(* Logix 5000 project; controller GEA_Test_Chamber vendor 1 type 14 code 196 rev 32.14; software revision 32.04; part 8 of 11 *)
(* tags used below, declared in another part *)
   Act_Time : DINT[7];
   Actuators_OnOff_Heater : BOOL;
   bPulse10Hz : BOOL;
   bPulse1Hz : BOOL;
   Counter : COUNTER[20];
   DRK375_Flow_Change : BOOL;
   DRK375_Flow_InRange : BOOL;
   DRK375_Temp_Change : BOOL;
   DRK375_Temp_InRange : BOOL;
   Flow_Change_Step : INT;
   FVIR_Water_DRK375_Error : REAL;
   Heater_OnOff : BOOL;
   LDO_DRK375_Start : BOOL;
   LDO_LabView_Comm_OK : BOOL;
   LDO_Step : INT;
   LDO_TestFlow : BOOL;
   LDO_Timer_Delay : TIMER[30];
   LDO_Water_float : REAL;
   LDO_Water_Flow_DRK375_REG : REAL;
   LDO_Water_Flow_DRK375_SP : INT;
   LDO_Water_SP_float : REAL;
   LDO_Water_Temp_DRK375_SP : INT;
   LDO_Water_Temp_float : REAL;
   LDO_Water_Temp_SP_float : REAL;
   LDO_WaterHeater_Step : INT;
   New_Time : BOOL;
   ONS : BOOL[32];
   puls_start : BOOL;
   puls_stop : BOOL;
   Pulse : BOOL[32];
   T_Diff_WaterStep10 : T_DIFF;
   T_Diff_WaterStep20 : T_DIFF;
   T_Diff_WaterStep40 : T_DIFF;
   T_Diff_WaterStep50 : T_DIFF;
   T_Diff_WaterStep70 : T_DIFF;
   T_Diff_WaterStep80 : T_DIFF;
   Temp_Change_Step : INT;
   Timer_Delay : TIMER[30];
   Water_Flow_Calc_float : REAL;
   Water_Flow_DRK375 : INT;
   Water_Outlet_InRange_LDO : BOOL;
   Water_Step_10 : DINT[7];
   Water_Step_10_Done : BOOL;
   Water_Step_20 : DINT[7];
   Water_Step_20_Done : BOOL;
   Water_Step_401 : DINT[7];
   Water_Step_40_Done : BOOL;
   Water_Step_50 : DINT[7];
   Water_Step_50_Done : BOOL;
   Water_Step_70 : DINT[7];
   Water_Step_70_Done : BOOL;
   Water_Step_80 : DINT[7];
   Water_Step_80_Done : BOOL;
   Water_T_Diff_10 : DINT;
   Water_T_Diff_20 : DINT;
   Water_T_Diff_40 : DINT;
   Water_T_Diff_50 : DINT;
   Water_T_Diff_70 : DINT;
   Water_T_Diff_80 : DINT;
   Water_Temp_Calc_float : REAL;
   Water_Temp_DRK375 : INT;
   Water_Temp_DRK375_Last : REAL;
   Heater_Cnt : COUNTER;
   LDO_Error_MSG : INT;
   LDO_LabView_Control : INT;
   LDO_Water_Flow_DRK375_Float : REAL;
   LDO_Water_Temp_DRK375_Float : REAL;
   Output_LDO : Output_LDO;
   Water_Flow_DRK375_Last_Float : REAL;
(* LDO_Chamber, continued *)

ROUTINE LDO_Error_MSG   (* ladder *)
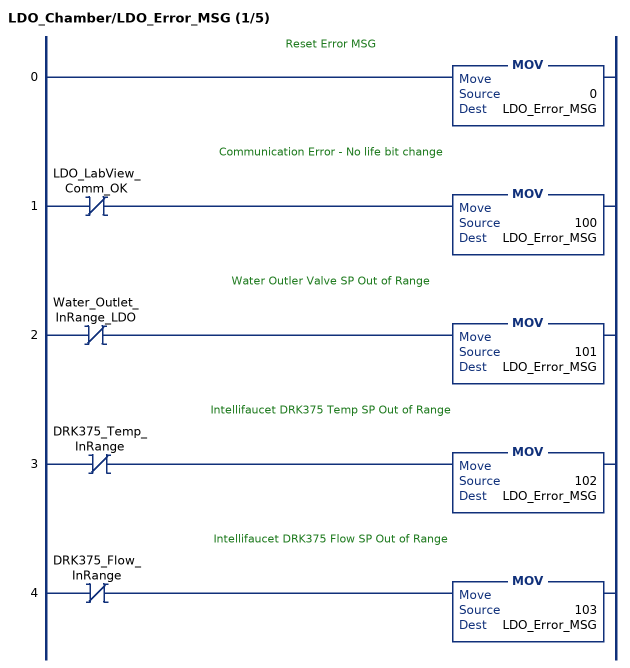
   // Reset Error MSG
   0: MOV(0,LDO_Error_MSG);
   // Communication Error - No life bit change
   1: XIO(LDO_LabView_Comm_OK)MOV(100,LDO_Error_MSG);
   // Water Outler Valve SP Out of Range
   2: XIO(Water_Outlet_InRange_LDO)MOV(101,LDO_Error_MSG);
   // Intellifaucet DRK375 Temp SP Out of Range
   3: XIO(DRK375_Temp_InRange)MOV(102,LDO_Error_MSG);
   // Intellifaucet DRK375 Flow SP Out of Range
   4: XIO(DRK375_Flow_InRange)MOV(103,LDO_Error_MSG);
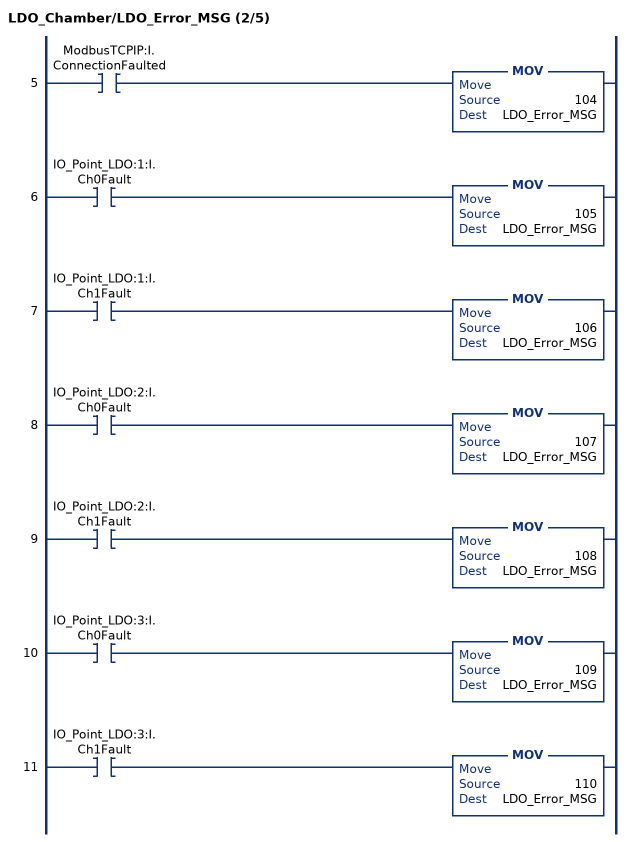
   5: XIC(ModbusTCPIP:I.ConnectionFaulted)MOV(104,LDO_Error_MSG);
   6: XIC(IO_Point_LDO:1:I.Ch0Fault)MOV(105,LDO_Error_MSG);
   7: XIC(IO_Point_LDO:1:I.Ch1Fault)MOV(106,LDO_Error_MSG);
   8: XIC(IO_Point_LDO:2:I.Ch0Fault)MOV(107,LDO_Error_MSG);
   9: XIC(IO_Point_LDO:2:I.Ch1Fault)MOV(108,LDO_Error_MSG);
   10: XIC(IO_Point_LDO:3:I.Ch0Fault)MOV(109,LDO_Error_MSG);
   11: XIC(IO_Point_LDO:3:I.Ch1Fault)MOV(110,LDO_Error_MSG);
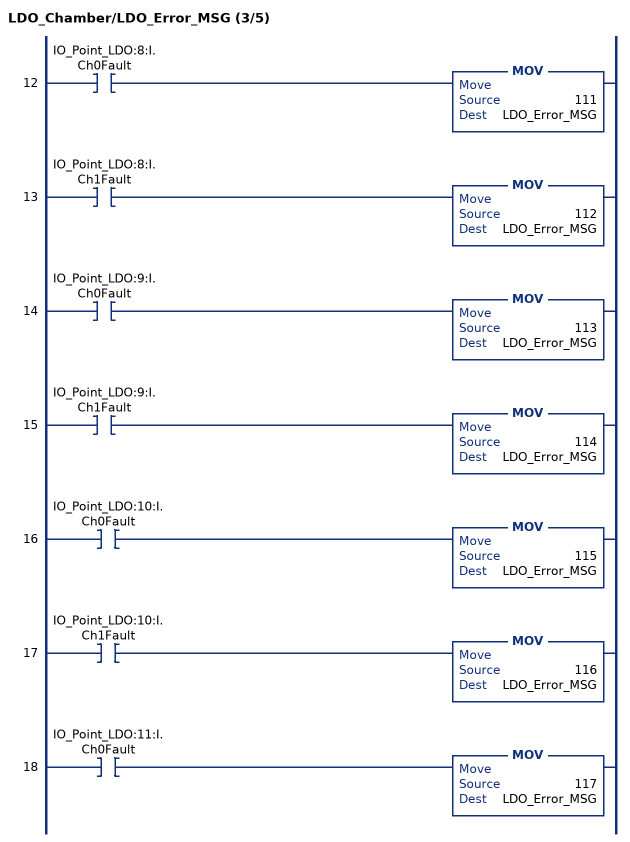
   12: XIC(IO_Point_LDO:8:I.Ch0Fault)MOV(111,LDO_Error_MSG);
   13: XIC(IO_Point_LDO:8:I.Ch1Fault)MOV(112,LDO_Error_MSG);
   14: XIC(IO_Point_LDO:9:I.Ch0Fault)MOV(113,LDO_Error_MSG);
   15: XIC(IO_Point_LDO:9:I.Ch1Fault)MOV(114,LDO_Error_MSG);
   16: XIC(IO_Point_LDO:10:I.Ch0Fault)MOV(115,LDO_Error_MSG);
   17: XIC(IO_Point_LDO:10:I.Ch1Fault)MOV(116,LDO_Error_MSG);
   18: XIC(IO_Point_LDO:11:I.Ch0Fault)MOV(117,LDO_Error_MSG);
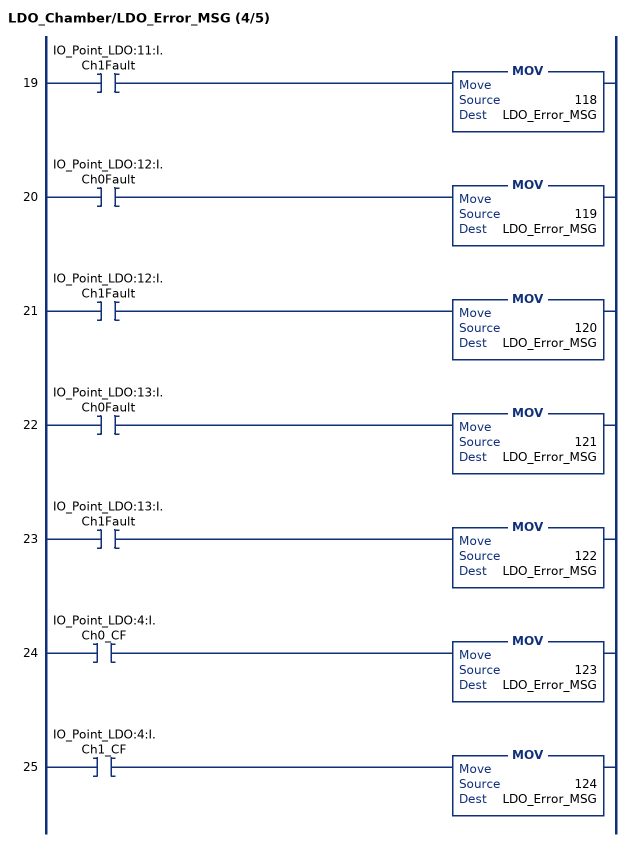
   19: XIC(IO_Point_LDO:11:I.Ch1Fault)MOV(118,LDO_Error_MSG);
   20: XIC(IO_Point_LDO:12:I.Ch0Fault)MOV(119,LDO_Error_MSG);
   21: XIC(IO_Point_LDO:12:I.Ch1Fault)MOV(120,LDO_Error_MSG);
   22: XIC(IO_Point_LDO:13:I.Ch0Fault)MOV(121,LDO_Error_MSG);
   23: XIC(IO_Point_LDO:13:I.Ch1Fault)MOV(122,LDO_Error_MSG);
   24: XIC(IO_Point_LDO:4:I.Ch0_CF)MOV(123,LDO_Error_MSG);
   25: XIC(IO_Point_LDO:4:I.Ch1_CF)MOV(124,LDO_Error_MSG);
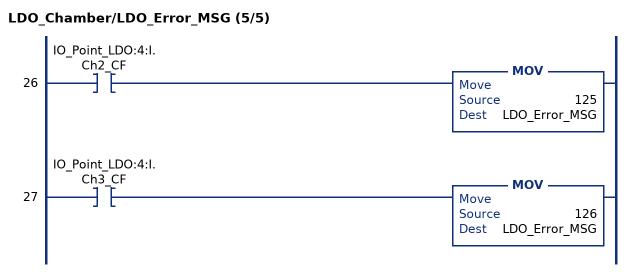
   26: XIC(IO_Point_LDO:4:I.Ch2_CF)MOV(125,LDO_Error_MSG);
   27: XIC(IO_Point_LDO:4:I.Ch3_CF)MOV(126,LDO_Error_MSG);
END_ROUTINE

ROUTINE LDO_Heater_OnOff   (* ladder *)
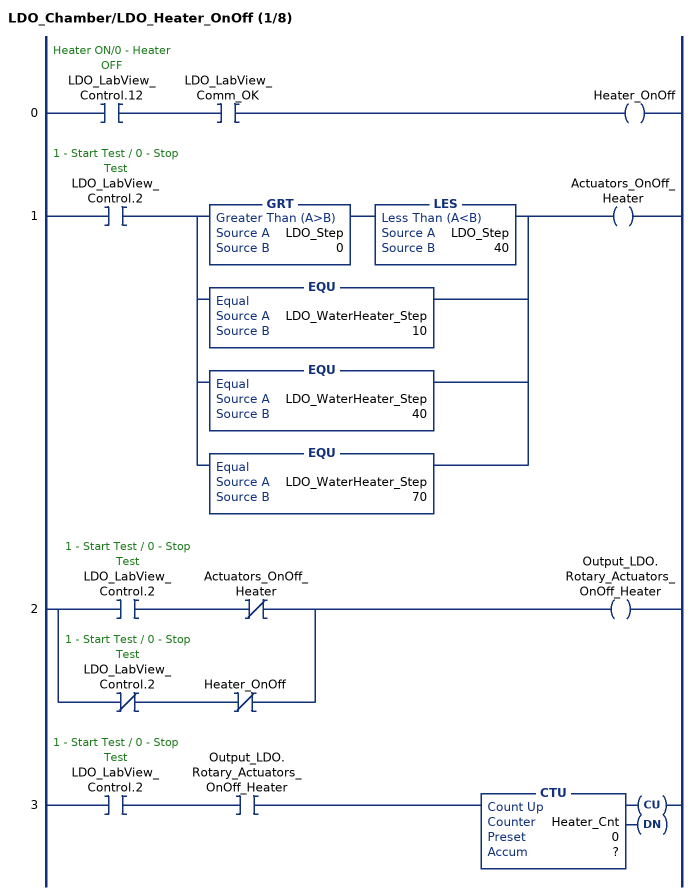
   0: XIC(LDO_LabView_Control.12)XIC(LDO_LabView_Comm_OK)OTE(Heater_OnOff);
   1: XIC(LDO_LabView_Control.2)[GRT(LDO_Step,0) LES(LDO_Step,40) ,EQU(LDO_WaterHeater_Step,10) ,EQU(LDO_WaterHeater_Step,40) ,EQU(LDO_WaterHeater_Step,70) ]OTE(Actuators_OnOff_Heater);
   2: [XIC(LDO_LabView_Control.2) XIO(Actuators_OnOff_Heater) ,XIO(LDO_LabView_Control.2) XIO(Heater_OnOff) ]OTE(Output_LDO.Rotary_Actuators_OnOff_Heater);
   3: XIC(LDO_LabView_Control.2)XIC(Output_LDO.Rotary_Actuators_OnOff_Heater)CTU(Heater_Cnt,?,?);
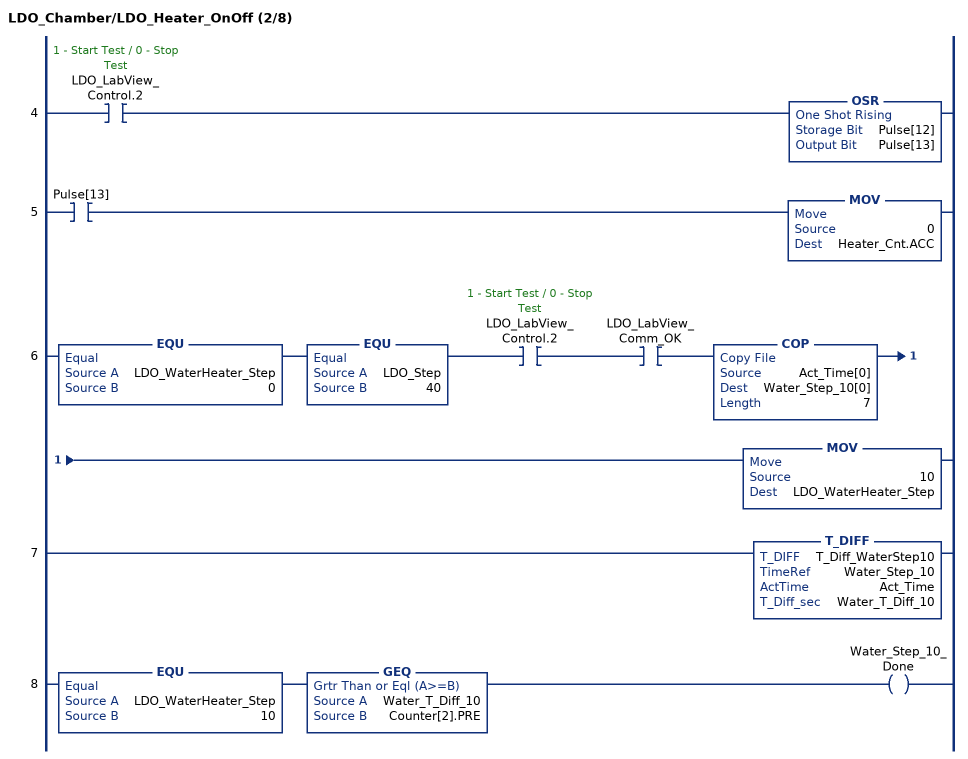
   4: XIC(LDO_LabView_Control.2)OSR(Pulse[12],Pulse[13]);
   5: XIC(Pulse[13])MOV(0,Heater_Cnt.ACC);
   6: EQU(LDO_WaterHeater_Step,0)EQU(LDO_Step,40)XIC(LDO_LabView_Control.2)XIC(LDO_LabView_Comm_OK)COP(Act_Time[0],Water_Step_10[0],7)MOV(10,LDO_WaterHeater_Step);
   7: T_DIFF(T_Diff_WaterStep10,Water_Step_10,Act_Time,Water_T_Diff_10);
   8: EQU(LDO_WaterHeater_Step,10)GEQ(Water_T_Diff_10,Counter[2].PRE)OTE(Water_Step_10_Done);
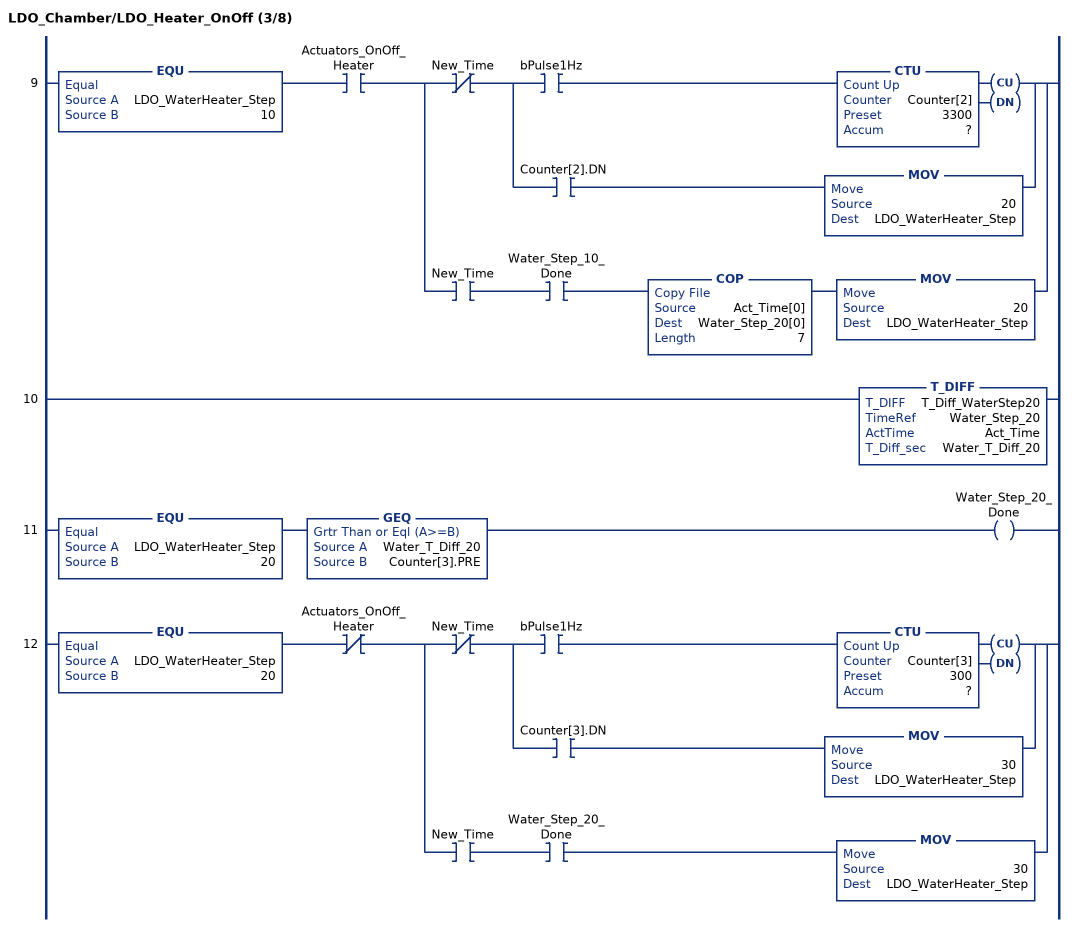
   9: EQU(LDO_WaterHeater_Step,10)XIC(Actuators_OnOff_Heater)[XIO(New_Time) [XIC(bPulse1Hz) CTU(Counter[2],?,?) ,XIC(Counter[2].DN) MOV(20,LDO_WaterHeater_Step) ] ,XIC(New_Time) XIC(Water_Step_10_Done) COP(Act_Time[0],Water_Step_20[0],7) MOV(20,LDO_WaterHeater_Step) ];
   10: T_DIFF(T_Diff_WaterStep20,Water_Step_20,Act_Time,Water_T_Diff_20);
   11: EQU(LDO_WaterHeater_Step,20)GEQ(Water_T_Diff_20,Counter[3].PRE)OTE(Water_Step_20_Done);
   12: EQU(LDO_WaterHeater_Step,20)XIO(Actuators_OnOff_Heater)[XIO(New_Time) [XIC(bPulse1Hz) CTU(Counter[3],?,?) ,XIC(Counter[3].DN) MOV(30,LDO_WaterHeater_Step) ] ,XIC(New_Time) XIC(Water_Step_20_Done) MOV(30,LDO_WaterHeater_Step) ];
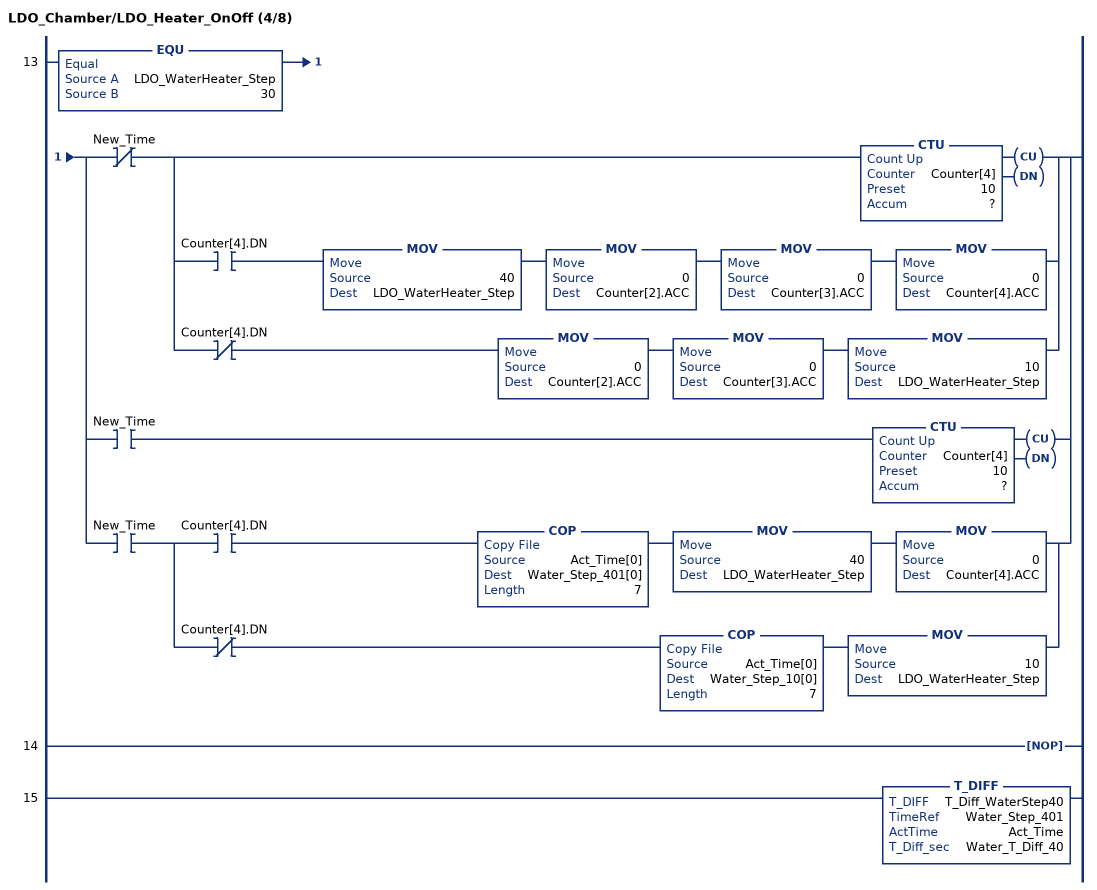
   13: EQU(LDO_WaterHeater_Step,30)[XIO(New_Time) [CTU(Counter[4],?,?) ,XIC(Counter[4].DN) MOV(40,LDO_WaterHeater_Step) MOV(0,Counter[2].ACC) MOV(0,Counter[3].ACC) MOV(0,Counter[4].ACC) ,XIO(Counter[4].DN) MOV(0,Counter[2].ACC) MOV(0,Counter[3].ACC) MOV(10,LDO_WaterHeater_Step) ] ,XIC(New_Time) CTU(Counter[4],?,?) ,XIC(New_Time) [XIC(Counter[4].DN) COP(Act_Time[0],Water_Step_401[0],7) MOV(40,LDO_WaterHeater_Step) MOV(0,Counter[4].ACC) ,XIO(Counter[4].DN) COP(Act_Time[0],Water_Step_10[0],7) MOV(10,LDO_WaterHeater_Step) ] ];
   14: NOP();
   15: T_DIFF(T_Diff_WaterStep40,Water_Step_401,Act_Time,Water_T_Diff_40);
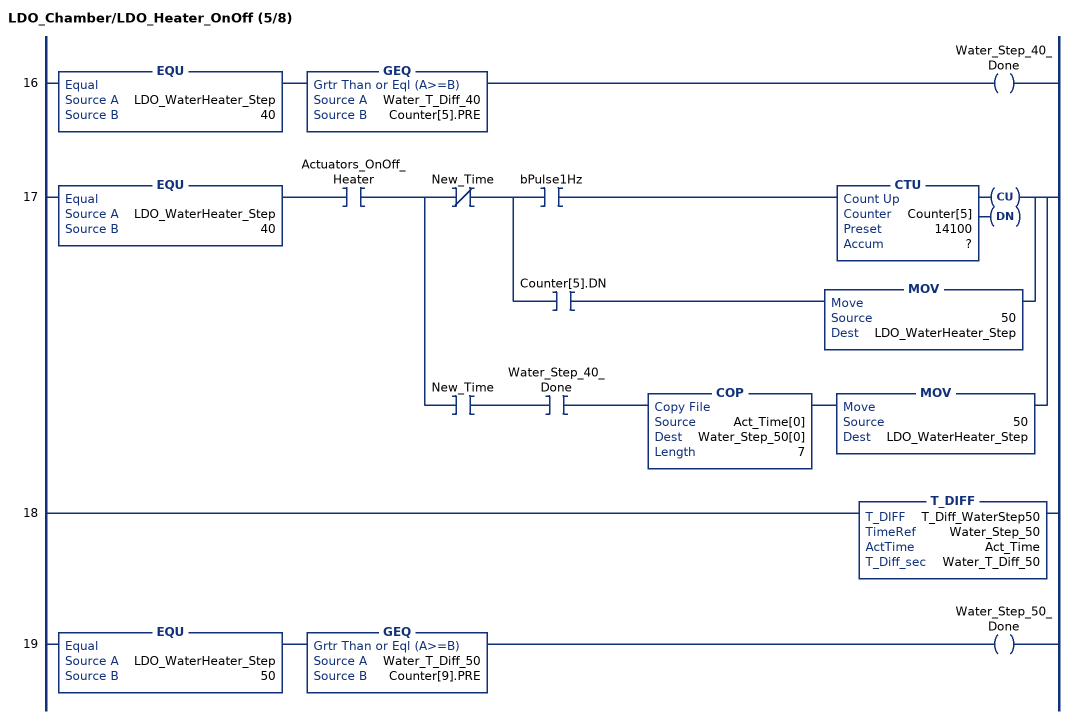
   16: EQU(LDO_WaterHeater_Step,40)GEQ(Water_T_Diff_40,Counter[5].PRE)OTE(Water_Step_40_Done);
   17: EQU(LDO_WaterHeater_Step,40)XIC(Actuators_OnOff_Heater)[XIO(New_Time) [XIC(bPulse1Hz) CTU(Counter[5],?,?) ,XIC(Counter[5].DN) MOV(50,LDO_WaterHeater_Step) ] ,XIC(New_Time) XIC(Water_Step_40_Done) COP(Act_Time[0],Water_Step_50[0],7) MOV(50,LDO_WaterHeater_Step) ];
   18: T_DIFF(T_Diff_WaterStep50,Water_Step_50,Act_Time,Water_T_Diff_50);
   19: EQU(LDO_WaterHeater_Step,50)GEQ(Water_T_Diff_50,Counter[9].PRE)OTE(Water_Step_50_Done);
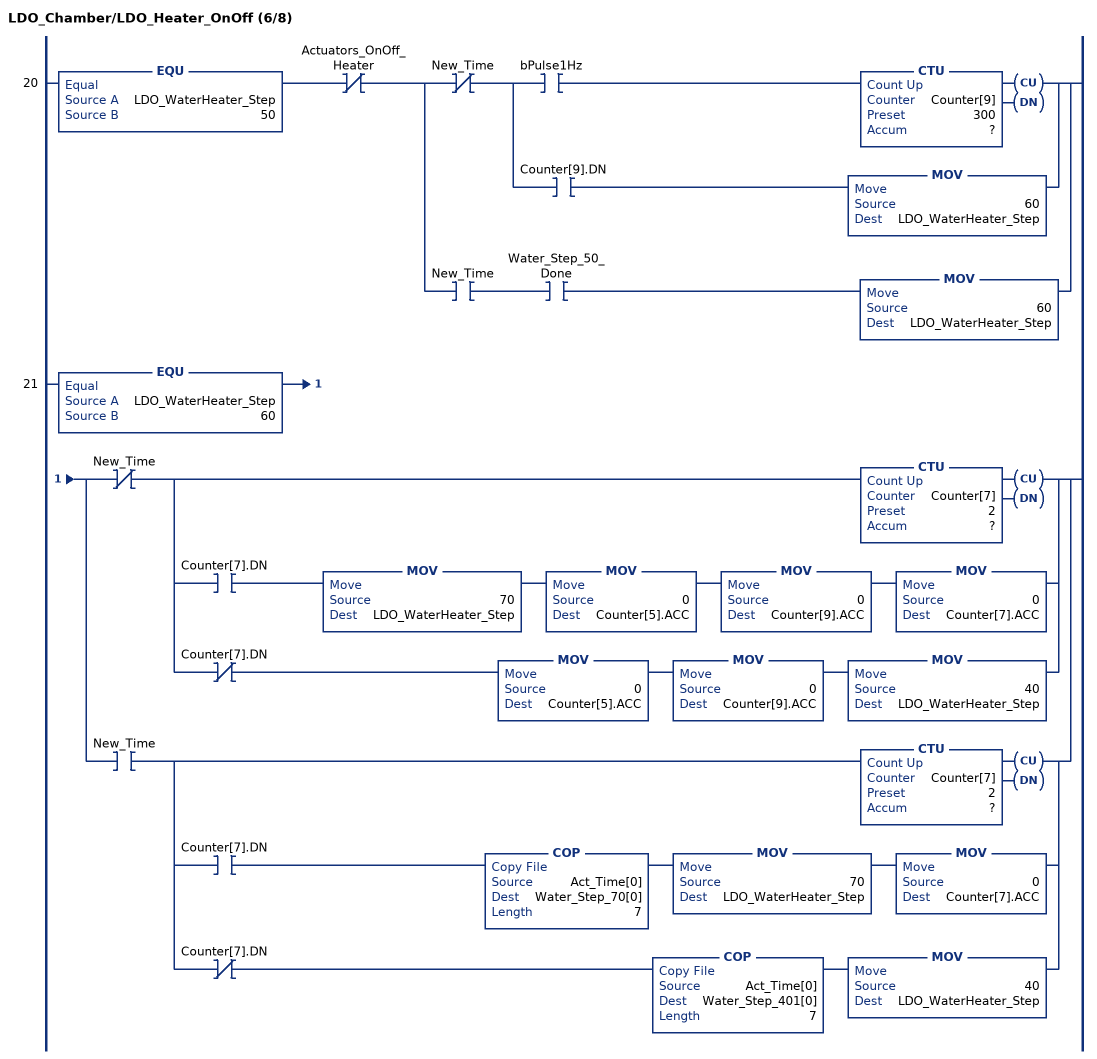
   20: EQU(LDO_WaterHeater_Step,50)XIO(Actuators_OnOff_Heater)[XIO(New_Time) [XIC(bPulse1Hz) CTU(Counter[9],?,?) ,XIC(Counter[9].DN) MOV(60,LDO_WaterHeater_Step) ] ,XIC(New_Time) XIC(Water_Step_50_Done) MOV(60,LDO_WaterHeater_Step) ];
   21: EQU(LDO_WaterHeater_Step,60)[XIO(New_Time) [CTU(Counter[7],?,?) ,XIC(Counter[7].DN) MOV(70,LDO_WaterHeater_Step) MOV(0,Counter[5].ACC) MOV(0,Counter[9].ACC) MOV(0,Counter[7].ACC) ,XIO(Counter[7].DN) MOV(0,Counter[5].ACC) MOV(0,Counter[9].ACC) MOV(40,LDO_WaterHeater_Step) ] ,XIC(New_Time) [CTU(Counter[7],?,?) ,XIC(Counter[7].DN) COP(Act_Time[0],Water_Step_70[0],7) MOV(70,LDO_WaterHeater_Step) MOV(0,Counter[7].ACC) ,XIO(Counter[7].DN) COP(Act_Time[0],Water_Step_401[0],7) MOV(40,LDO_WaterHeater_Step) ] ];
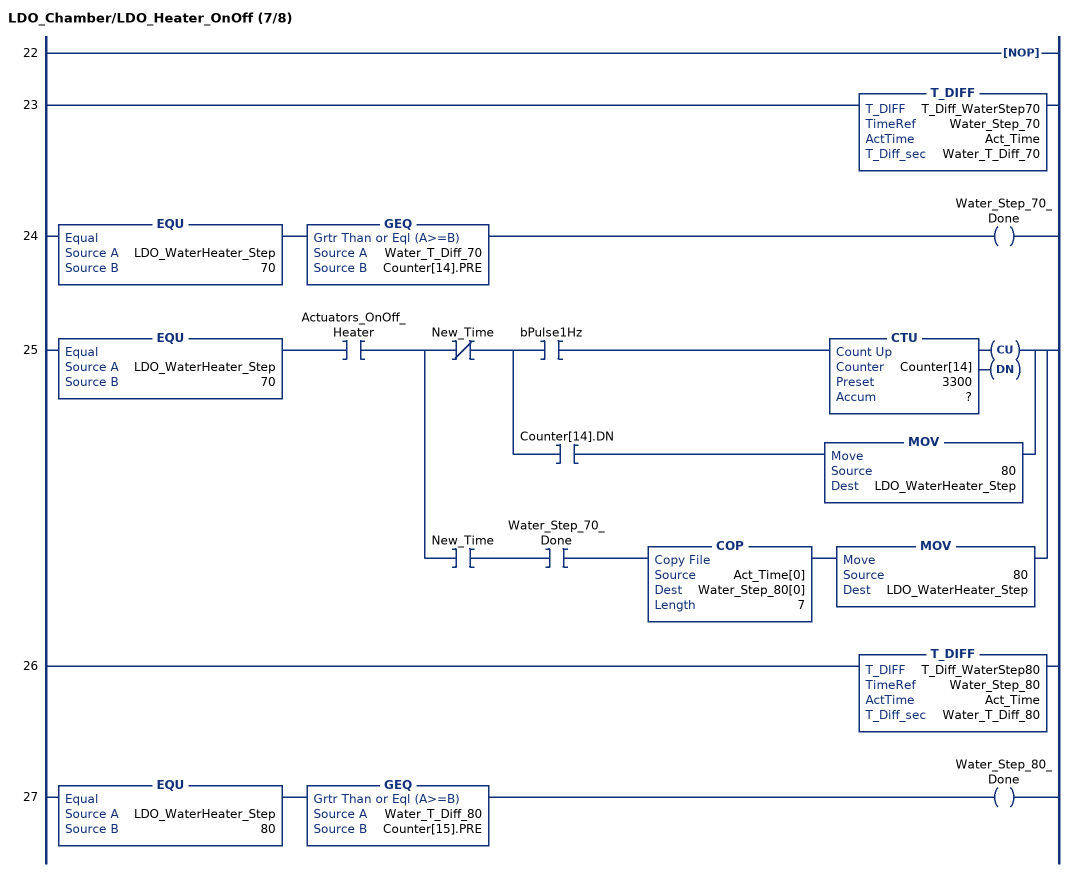
   22: NOP();
   23: T_DIFF(T_Diff_WaterStep70,Water_Step_70,Act_Time,Water_T_Diff_70);
   24: EQU(LDO_WaterHeater_Step,70)GEQ(Water_T_Diff_70,Counter[14].PRE)OTE(Water_Step_70_Done);
   25: EQU(LDO_WaterHeater_Step,70)XIC(Actuators_OnOff_Heater)[XIO(New_Time) [XIC(bPulse1Hz) CTU(Counter[14],?,?) ,XIC(Counter[14].DN) MOV(80,LDO_WaterHeater_Step) ] ,XIC(New_Time) XIC(Water_Step_70_Done) COP(Act_Time[0],Water_Step_80[0],7) MOV(80,LDO_WaterHeater_Step) ];
   26: T_DIFF(T_Diff_WaterStep80,Water_Step_80,Act_Time,Water_T_Diff_80);
   27: EQU(LDO_WaterHeater_Step,80)GEQ(Water_T_Diff_80,Counter[15].PRE)OTE(Water_Step_80_Done);
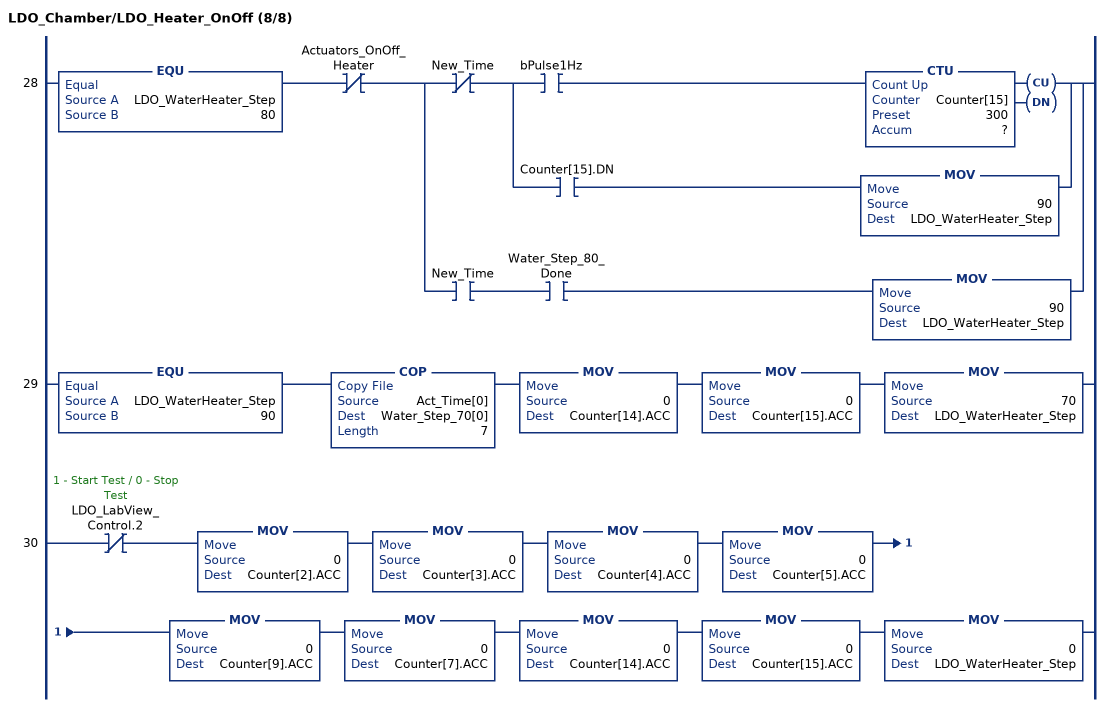
   28: EQU(LDO_WaterHeater_Step,80)XIO(Actuators_OnOff_Heater)[XIO(New_Time) [XIC(bPulse1Hz) CTU(Counter[15],?,?) ,XIC(Counter[15].DN) MOV(90,LDO_WaterHeater_Step) ] ,XIC(New_Time) XIC(Water_Step_80_Done) MOV(90,LDO_WaterHeater_Step) ];
   29: EQU(LDO_WaterHeater_Step,90)COP(Act_Time[0],Water_Step_70[0],7)MOV(0,Counter[14].ACC)MOV(0,Counter[15].ACC)MOV(70,LDO_WaterHeater_Step);
   30: XIO(LDO_LabView_Control.2)MOV(0,Counter[2].ACC)MOV(0,Counter[3].ACC)MOV(0,Counter[4].ACC)MOV(0,Counter[5].ACC)MOV(0,Counter[9].ACC)MOV(0,Counter[7].ACC)MOV(0,Counter[14].ACC)MOV(0,Counter[15].ACC)MOV(0,LDO_WaterHeater_Step);
END_ROUTINE

ROUTINE LDO_Intellfaucet_Control   (* ladder *)
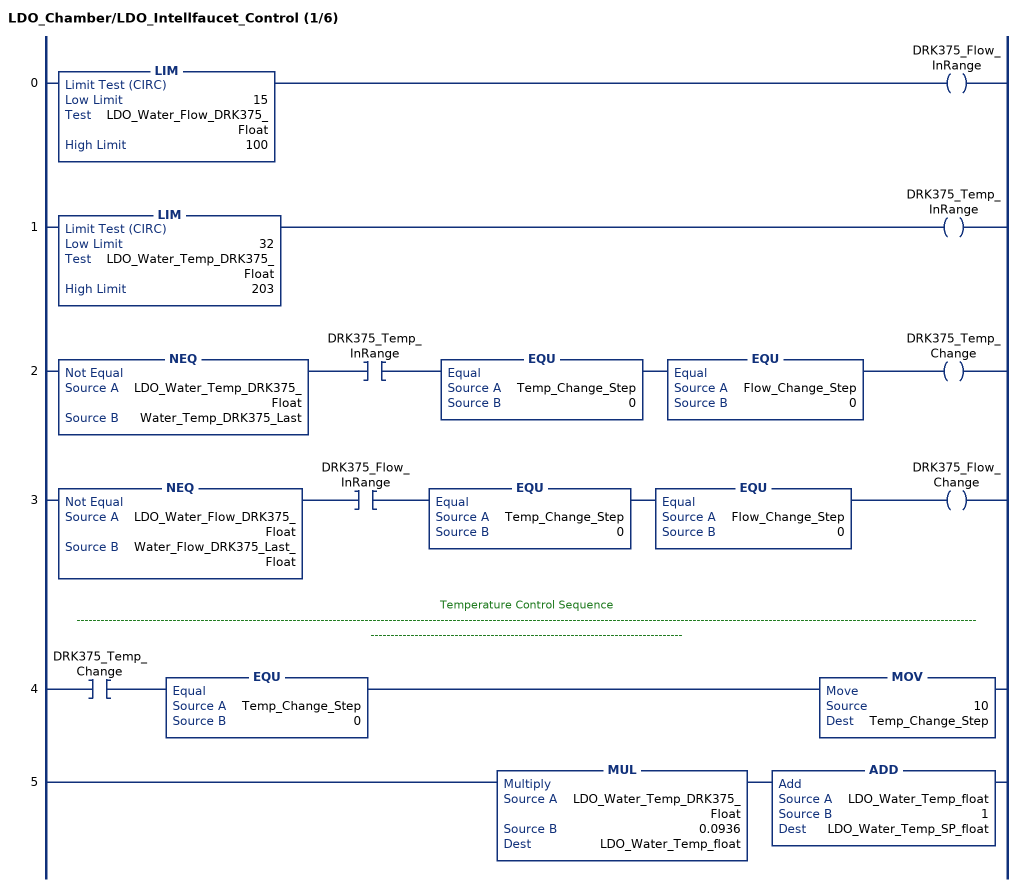
   0: LIM(15,LDO_Water_Flow_DRK375_Float,100)OTE(DRK375_Flow_InRange);
   1: LIM(32,LDO_Water_Temp_DRK375_Float,203)OTE(DRK375_Temp_InRange);
   2: NEQ(LDO_Water_Temp_DRK375_Float,Water_Temp_DRK375_Last)XIC(DRK375_Temp_InRange)EQU(Temp_Change_Step,0)EQU(Flow_Change_Step,0)OTE(DRK375_Temp_Change);
   3: NEQ(LDO_Water_Flow_DRK375_Float,Water_Flow_DRK375_Last_Float)XIC(DRK375_Flow_InRange)EQU(Temp_Change_Step,0)EQU(Flow_Change_Step,0)OTE(DRK375_Flow_Change);
   // Temperature Control Sequence
   // ---------------------------------------------------------------------------------------------------------------------------------------------------------------------------------------------------------------------------------------------------------------------------------------------------------------
   4: XIC(DRK375_Temp_Change)EQU(Temp_Change_Step,0)MOV(10,Temp_Change_Step);
   5: MUL(LDO_Water_Temp_DRK375_Float,0.0936,LDO_Water_Temp_float)ADD(LDO_Water_Temp_float,1,LDO_Water_Temp_SP_float);
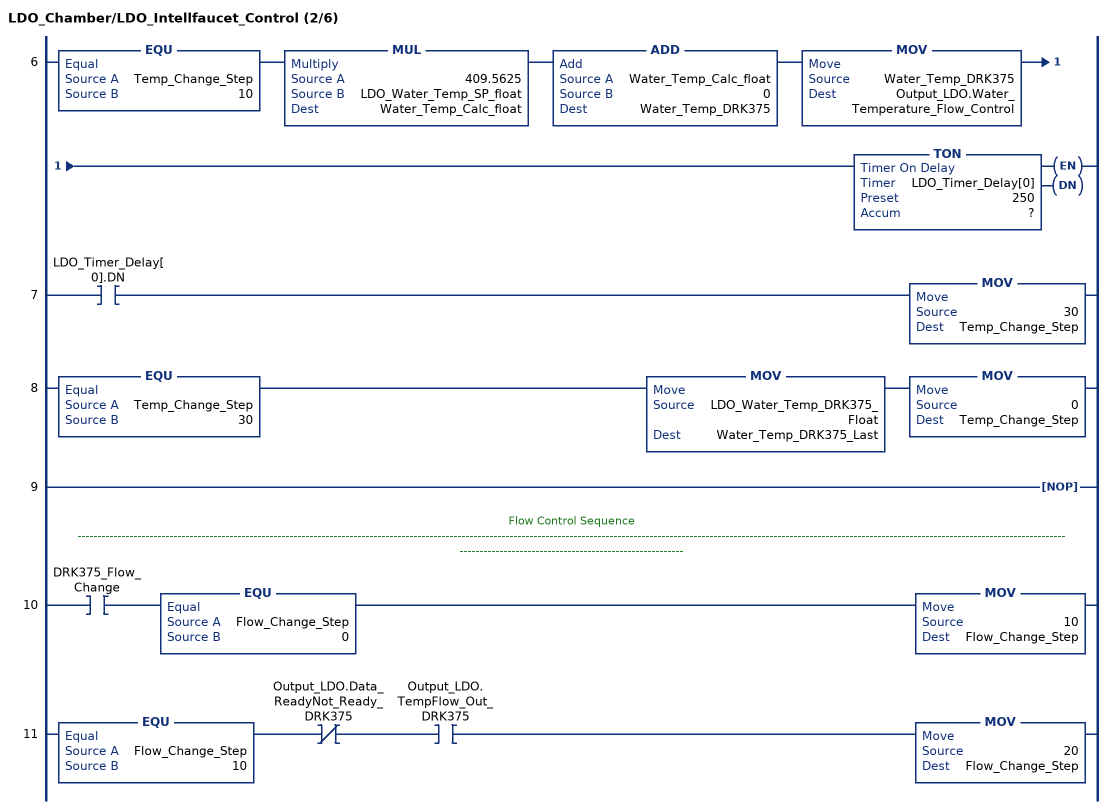
   6: EQU(Temp_Change_Step,10)MUL(409.5625,LDO_Water_Temp_SP_float,Water_Temp_Calc_float)ADD(Water_Temp_Calc_float,0,Water_Temp_DRK375)MOV(Water_Temp_DRK375,Output_LDO.Water_Temperature_Flow_Control)TON(LDO_Timer_Delay[0],?,?);
   7: XIC(LDO_Timer_Delay[0].DN)MOV(30,Temp_Change_Step);
   8: EQU(Temp_Change_Step,30)MOV(LDO_Water_Temp_DRK375_Float,Water_Temp_DRK375_Last)MOV(0,Temp_Change_Step);
   9: NOP();
   // Flow Control Sequence
   // ---------------------------------------------------------------------------------------------------------------------------------------------------------------------------------------------------------------------------------------------------------------------------------------------------------------
   10: XIC(DRK375_Flow_Change)EQU(Flow_Change_Step,0)MOV(10,Flow_Change_Step);
   11: EQU(Flow_Change_Step,10)XIO(Output_LDO.Data_ReadyNot_Ready_DRK375)XIC(Output_LDO.TempFlow_Out_DRK375)MOV(20,Flow_Change_Step);
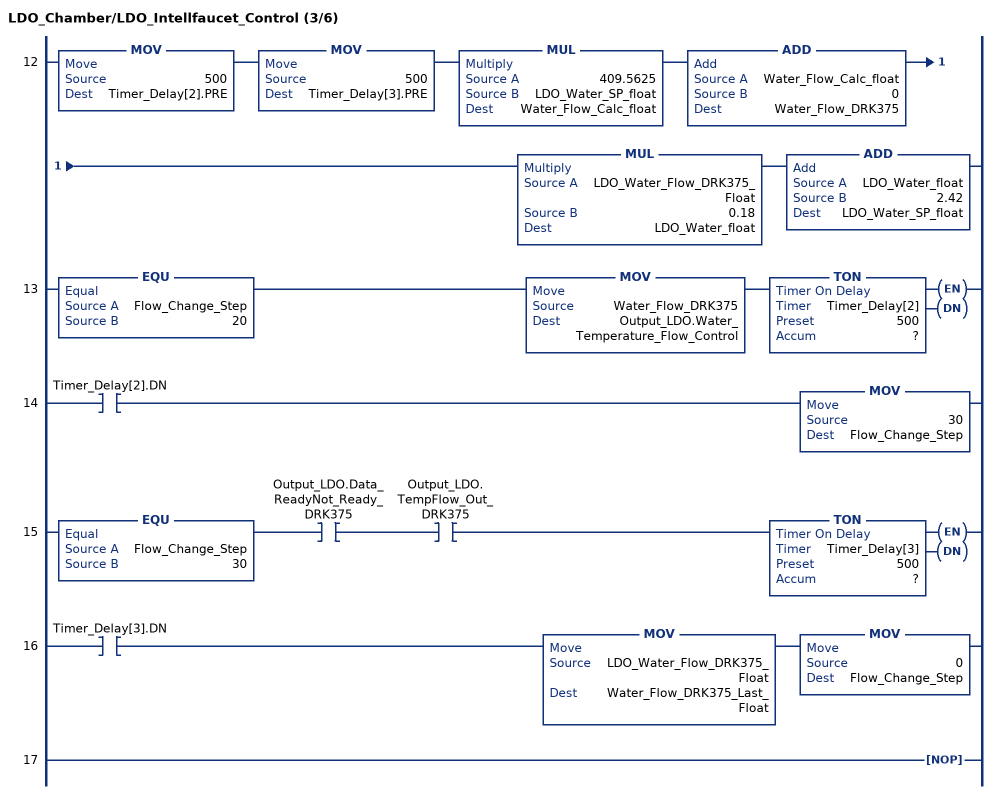
   12: MOV(500,Timer_Delay[2].PRE)MOV(500,Timer_Delay[3].PRE)MUL(409.5625,LDO_Water_SP_float,Water_Flow_Calc_float)ADD(Water_Flow_Calc_float,0,Water_Flow_DRK375)MUL(LDO_Water_Flow_DRK375_Float,0.18,LDO_Water_float)ADD(LDO_Water_float,2.42,LDO_Water_SP_float);
   13: EQU(Flow_Change_Step,20)MOV(Water_Flow_DRK375,Output_LDO.Water_Temperature_Flow_Control)TON(Timer_Delay[2],?,?);
   14: XIC(Timer_Delay[2].DN)MOV(30,Flow_Change_Step);
   15: EQU(Flow_Change_Step,30)XIC(Output_LDO.Data_ReadyNot_Ready_DRK375)XIC(Output_LDO.TempFlow_Out_DRK375)TON(Timer_Delay[3],?,?);
   16: XIC(Timer_Delay[3].DN)MOV(LDO_Water_Flow_DRK375_Float,Water_Flow_DRK375_Last_Float)MOV(0,Flow_Change_Step);
   17: NOP();
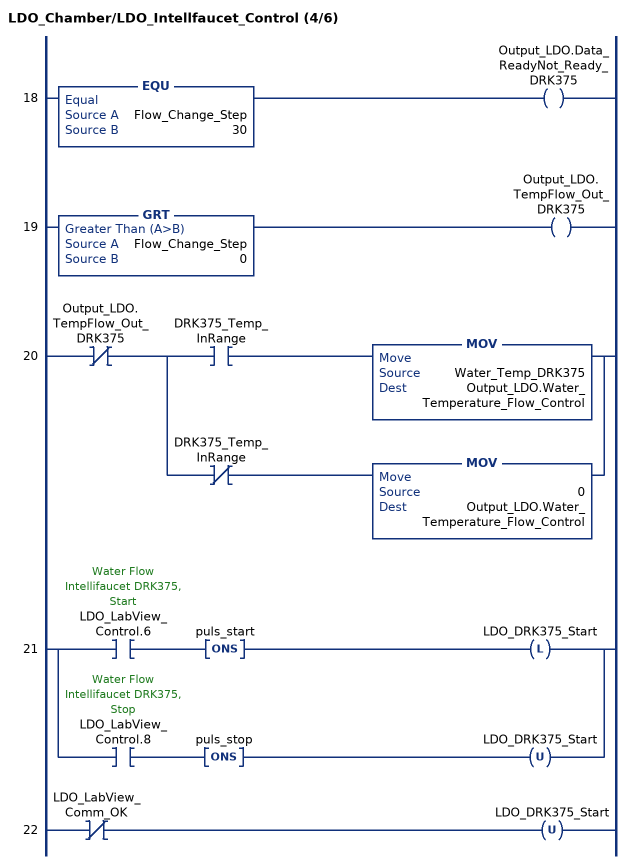
   18: EQU(Flow_Change_Step,30)OTE(Output_LDO.Data_ReadyNot_Ready_DRK375);
   19: GRT(Flow_Change_Step,0)OTE(Output_LDO.TempFlow_Out_DRK375);
   20: XIO(Output_LDO.TempFlow_Out_DRK375)[XIC(DRK375_Temp_InRange) MOV(Water_Temp_DRK375,Output_LDO.Water_Temperature_Flow_Control) ,XIO(DRK375_Temp_InRange) MOV(0,Output_LDO.Water_Temperature_Flow_Control) ];
   21: [XIC(LDO_LabView_Control.6) ONS(puls_start) OTL(LDO_DRK375_Start) ,XIC(LDO_LabView_Control.8) ONS(puls_stop) OTU(LDO_DRK375_Start) ];
   22: XIO(LDO_LabView_Comm_OK)OTU(LDO_DRK375_Start);
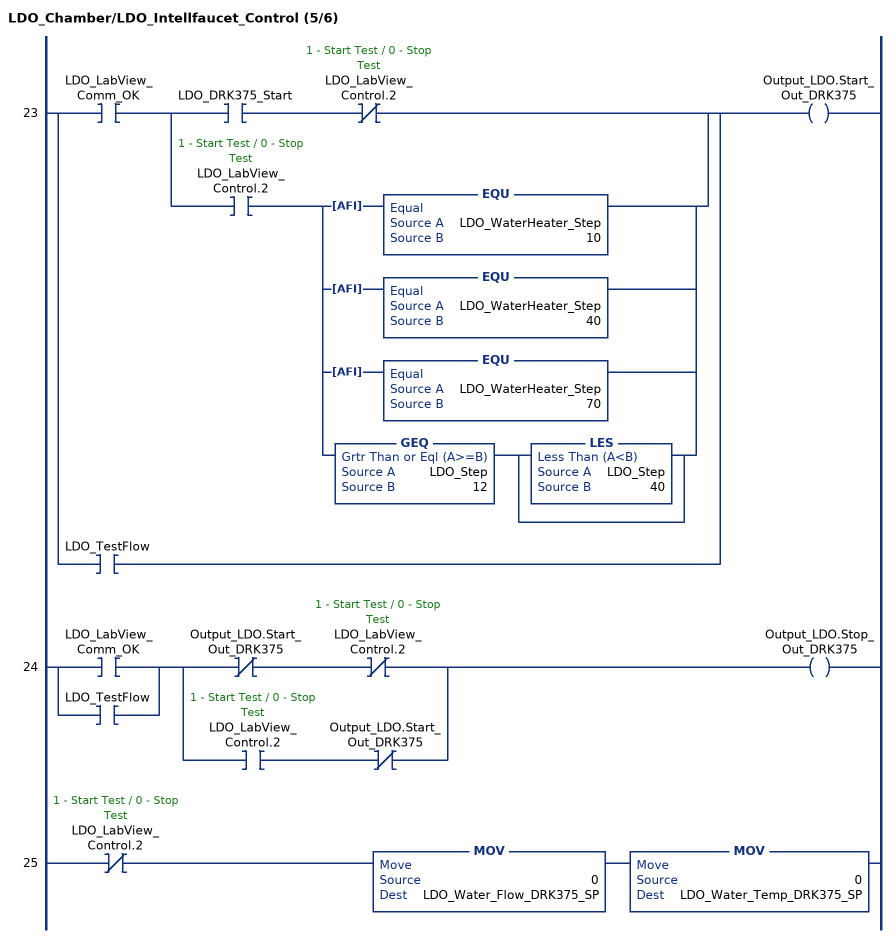
   23: [XIC(LDO_LabView_Comm_OK) [XIC(LDO_DRK375_Start) XIO(LDO_LabView_Control.2) ,XIC(LDO_LabView_Control.2) [AFI() EQU(LDO_WaterHeater_Step,10) ,AFI() EQU(LDO_WaterHeater_Step,40) ,AFI() EQU(LDO_WaterHeater_Step,70) ,GEQ(LDO_Step,12) [LES(LDO_Step,40) ,] ] ] ,XIC(LDO_TestFlow) ]OTE(Output_LDO.Start_Out_DRK375);
   24: [XIC(LDO_LabView_Comm_OK) ,XIC(LDO_TestFlow) ][XIO(Output_LDO.Start_Out_DRK375) XIO(LDO_LabView_Control.2) ,XIC(LDO_LabView_Control.2) XIO(Output_LDO.Start_Out_DRK375) ]OTE(Output_LDO.Stop_Out_DRK375);
   25: XIO(LDO_LabView_Control.2)MOV(0,LDO_Water_Flow_DRK375_SP)MOV(0,LDO_Water_Temp_DRK375_SP);
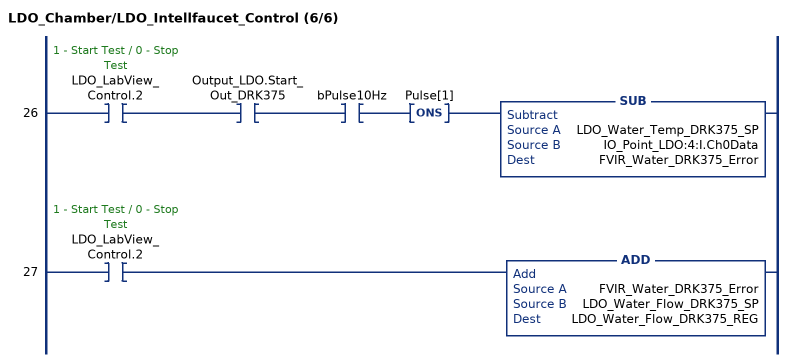
   26: XIC(LDO_LabView_Control.2)XIC(Output_LDO.Start_Out_DRK375)XIC(bPulse10Hz)ONS(Pulse[1])SUB(LDO_Water_Temp_DRK375_SP,IO_Point_LDO:4:I.Ch0Data,FVIR_Water_DRK375_Error);
   27: XIC(LDO_LabView_Control.2)ADD(FVIR_Water_DRK375_Error,LDO_Water_Flow_DRK375_SP,LDO_Water_Flow_DRK375_REG);
END_ROUTINE
